(* CODESYS project Elevator_student_1.project

Project tree, tasks and I/O mapping:
  Device : CODESYS Control Win V3, 3S - Smart Software Solutions GmbH, version 3.5.17.10
    application Application
      libraries: Standard, * (System); VisuDialogs, * (System); Util, * (System)
      task MainTask (cyclic, interval t#10ms, priority 1) calls Model, PLC_PRG
      program Model [ST]
      visualisation Visualization
      global variables GVL
      program PLC_PRG [ST]
      function block StartMotor [ST]
      function block DoorOpenClose [FBD]
  text list GlobalTextList
*)

// Device/Application/GVL
VAR_GLOBAL
	// Sensors:
	onfloor0:BOOL;		// Elevator at floor 0
	onfloor1:BOOL;		// Elevator at floor 1
	onfloor2:BOOL;		// Elevator at floor 2
	doorclosed0:BOOL;	// Doors at floor 0 are closed
	doorclosed1:BOOL;	// Doors at floor 1 are closed
	doorclosed2:BOOL;	// Doors at floor 2 are closed *)
	button0:BOOL;		// Call button at floor 0
	button1:BOOL;		// Call button at floor 1
	button2:BOOL;		// Call button at floor 2
	call0:BOOL;			// Request floor 0 from inside the cabin 
	call1:BOOL;			// Request floor 1 from inside the cabin
	call2:BOOL;			// Request floor 2 from inside the cabin
	
	// Actuators:
	up:BOOL;			// Control the elevator to go up
	down:BOOL;			// Control the elevator to go down
	open0:BOOL;			// Open the doors at floor 0
	open1:BOOL;			// Open the doors at floor 1
	open2:BOOL;			// Open the doors at floor 2
	
	// Other variables:
	go:BOOL;
	x:INT;				// Next destination floor number
END_VAR

// Device/Application/Model
PROGRAM Model

VAR CONSTANT
	// Define following variables as required
	maxSpeedLift :REAL := 0.5;
	accLift :REAL := 0.25;
	speedDoor :REAL := 0.5;
	cycleTime :DWORD := 10;
END_VAR

VAR
	// Following variables are inputs to the model
	motorUp :BOOL;
	motorDown :BOOL;
	door0 :BOOL;
	door1 :BOOL;
	door2 :BOOL;
	///////////////////////////////////////////////
	// Following variables are outpus from the model
	buttonFloor0: BOOL;
	buttonFloor1: BOOL;
	buttonFloor2: BOOL;
	requestFloor0 :BOOL;
	requestFloor1 :BOOL;
	requestFloor2 :BOOL;
	elevatorAtFloor0 :BOOL;
	elevatorAtFloor1 :BOOL;
	elevatorAtFloor2 :BOOL;
	door0Closed :BOOL;
	door1Closed :BOOL;
	door2Closed :BOOL;
	////////////////////////////////////////////
	elevatorPos :REAL :=30.0;
	speedLift :REAL := 0.0;
	doIntegral :INTEGRAL;
	door0LeftPos :REAL :=0.0;
	door0RightPos :REAL :=0.0;
	door1LeftPos :REAL :=0.0;
	door1RightPos :REAL :=0.0;
	door2LeftPos :REAL :=0.0;
	door2RightPos :REAL :=0.0;
	elevatorAtFloor :INT :=2;
	floor0 :BOOL;
	floor1 :BOOL;
	floor2 :BOOL;
	heightSensor :REAL := 0.0; // Output the height of the cabin.
END_VAR

// Definition of the inputs to the model, which correspond to the outputs from the controller.
motorUp := GVL.up;
motorDown := GVL.down;
door0 := GVL.open0;
door1 := GVL.open1;
door2 := GVL.open2;

// Control of the elevator
// First calculate its speed
IF motorUp OR motorDown THEN
	doIntegral(IN:=accLift,TM:=cycleTime,RESET:= NOT(motorUp OR motorDown),OUT=>speedLift);
ELSE
	doIntegral(RESET:=TRUE);
	speedLift := 0.0;
END_IF
// Limit the speed
IF (speedLift > maxSpeedLift) THEN
	speedLift := maxSpeedLift;
END_IF

// Then apply the speed if commanded
IF motorUp AND elevatorPos > 0.0 THEN
	elevatorPos := elevatorPos - speedLift;
END_IF

IF motorDown AND elevatorPos < 440.0 THEN
	elevatorPos := elevatorPos + speedLift;
END_IF

// Control of doors at floor 0. Doors are mirrored
IF door0 AND door0LeftPos > -50.0 THEN
	door0LeftPos := door0LeftPos - speedDoor;
	door0RightPos := - door0LeftPos;
END_IF
IF NOT(door0) AND door0LeftPos < 0.0 THEN
	door0LeftPos := door0LeftPos + speedDoor;
	door0RightPos := - door0LeftPos;
END_IF

// Control of doors at floor 1
IF door1 AND door1LeftPos > -50.0 THEN
	door1LeftPos := door1LeftPos - speedDoor;
	door1RightPos := - door1LeftPos;
END_IF
IF NOT(door1) AND door1LeftPos < 0.0 THEN
	door1LeftPos := door1LeftPos + speedDoor;
	door1RightPos := - door1LeftPos;
END_IF

// Control of doors at floor 2
IF door2 AND door2LeftPos > -50.0 THEN
	door2LeftPos := door2LeftPos - speedDoor;
	door2RightPos := - door2LeftPos;
END_IF
IF NOT(door2) AND door2LeftPos < 0.0 THEN
	door2LeftPos := door2LeftPos + speedDoor;
	door2RightPos := - door2LeftPos;
END_IF

// Status sensors whether the doors are closed or not
IF door0LeftPos < 0.0 THEN
	door0Closed := FALSE;
ELSE
	door0Closed := TRUE;
END_IF
IF door1LeftPos < 0.0 THEN
	door1Closed := FALSE;
ELSE
	door1Closed := TRUE;
END_IF
IF door2LeftPos < 0.0 THEN
	door2Closed := FALSE;
ELSE
	door2Closed := TRUE;
END_IF

// Determine floor number of elevator
IF elevatorPos < 30.5 THEN
	elevatorAtFloor := 2;
	elevatorAtFloor2 := TRUE;
	elevatorAtFloor0 := FALSE;
	elevatorAtFloor1 := FALSE;
ELSIF (elevatorPos  > 224.5) AND (elevatorPos < 225.5) THEN
	elevatorAtFloor := 1;
	elevatorAtFloor1 := TRUE;
	elevatorAtFloor0 := FALSE;
	elevatorAtFloor2 := FALSE;
ELSIF elevatorPos > 418.5 THEN
	elevatorAtFloor := 0;
	elevatorAtFloor0 := TRUE;
	elevatorAtFloor1 := FALSE;
	elevatorAtFloor2 := FALSE;
ELSE
	elevatorAtFloor2 := FALSE;
	elevatorAtFloor0 := FALSE;
	elevatorAtFloor1 := FALSE;	
END_IF

// Used to mantain the buttons state (visuzalization is a tap, hence a flip/flop is
// implemented here in order to mantain the status of the button and the "light".
IF floor0 THEN
	buttonFloor0 := TRUE;
END_IF
IF floor1 THEN
	buttonFloor1 := TRUE;
END_IF
IF floor2 THEN
	buttonFloor2 := TRUE;
END_IF

// Reset function for the request button. If the cabin is at the same floor and doors are opened,
// reset request of the floor
IF (requestFloor0 OR buttonFloor0) AND elevatorAtFloor0 AND (door0LeftPos < -49.5) THEN
	requestFloor0 := FALSE;
	buttonFloor0 := FALSE;
END_IF
IF (requestFloor1 OR buttonFloor1) AND elevatorAtFloor1 AND (door1LeftPos < -49.5) THEN
	requestFloor1 := FALSE;
	buttonFloor1 := FALSE;
END_IF
IF (requestFloor2 OR buttonFloor2) AND elevatorAtFloor2 AND (door2LeftPos < -49.5) THEN
	requestFloor2 := FALSE;
	buttonFloor2 := FALSE;
END_IF

// Extra functionality: the following code provides the reading of an analog sensor measuring the 
// height position of the elevator. It ouputs a value between 0..2 in normal conditions (i.e. the
// elevator does not go below o or over 2). If the elevator is driven below ground level, a minus
// sign number will be output. In case the elevator is driven over the second floor, a number
// higher than 2.0 will be output.
heightSensor := (419.0 - elevatorPos) / 389.0 * 2;

// Lastly, update outputs from the model, which correspond to the inputs of the controller.
GVL.button0 := buttonFloor0;
GVL.button1 := buttonFloor1;
GVL.button2 := buttonFloor2;
GVL.call0 := requestFloor0;
GVL.call1 := requestFloor1;
GVL.call2 := requestFloor2;
GVL.onfloor0 := elevatorAtFloor0;
GVL.onfloor1 := elevatorAtFloor1;
GVL.onfloor2 := elevatorAtFloor2;
GVL.doorclosed0 := door0Closed;
GVL.doorclosed1 := door1Closed;
GVL.doorclosed2 := door2Closed;

END_PROGRAM

// Device/Application/PLC_PRG
PROGRAM PLC_PRG
VAR
	startMoving:StartMotor;
	openClose:DoorOpenClose;
END_VAR

// Järjestelmätoiminto 1
gvl.go := TRUE;	// Yksikkötestausta varten
x := 0;			// Yksikkötestausta varten

WHILE gvl.go DO
	IF (gvl.onfloor0 AND x = 0) OR (gvl.onfloor1 AND x = 1) OR (gvl.onfloor2 AND x = 2) THEN;
		CASE gvl.x OF
		0:	gvl.open0 := TRUE;
			openClose();
			openClose.trigger := TRUE;
			gvl.open0 := openClose.output;
			
		1:	gvl.open1 := TRUE;
			openClose();
			openClose.trigger := TRUE;
			gvl.open1 := openClose.output;
			
		2:	gvl.open2 := TRUE;
			openClose();
			openClose.trigger := TRUE;
			gvl.open2 := openClose.output;
		END_CASE
		gvl.go := FALSE;
		RETURN;
	END_IF
	
	startMoving();
	Model();

	IF (NOT x = 1) AND gvl.onfloor1 AND (gvl.button1 OR gvl.call1) THEN
		gvl.up := FALSE;
		gvl.down := FALSE;
		gvl.open1 := TRUE;
		openClose();
		openClose.trigger := TRUE;
		gvl.open1 := openClose.output;
		gvl.call1 := FALSE;
		gvl.button1 := FALSE;
		startMoving();
		Model();
		openClose.trigger := FALSE;
	END_IF
		
	IF (x = 0 AND gvl.onfloor0) OR (x = 1 AND gvl.onfloor1) OR (x = 2 AND gvl.onfloor2) THEN
		gvl.up := FALSE;
		gvl.down := FALSE;
		CASE gvl.x OF
		0:	gvl.open0 := TRUE;
			openClose();
			openClose.trigger := TRUE;
			gvl.open0 := openClose.output;
			
		1:	gvl.open1 := TRUE;
			openClose();
			openClose.trigger := TRUE;
			gvl.open1 := openClose.output;
			
		2:	gvl.open2 := TRUE;  
			openClose();
			openClose.trigger := TRUE;
			gvl.open2 := openClose.output;	
		END_CASE
		gvl.go := FALSE;
	END_IF
	
	openClose.trigger := FALSE;
END_WHILE

END_PROGRAM

// Device/Application/StartMotor
FUNCTION_BLOCK StartMotor

IF gvl.onfloor0 AND (x = 1 OR x = 2) THEN;
	gvl.up := TRUE;
ELSIF gvl.onfloor2 AND (x = 0 OR x = 1) THEN;
	gvl.down := TRUE;
ELSIF gvl.onfloor1 AND x = 0 THEN;
	gvl.down := TRUE;
ELSIF gvl.onfloor1 AND x = 2 THEN;
	gvl.up := TRUE;
END_IF

END_FUNCTION_BLOCK

// Device/Application/DoorOpenClose
FUNCTION_BLOCK DoorOpenClose
VAR_INPUT
	trigger: BOOL;
	delay: TIME := T#1.5S;
END_VAR
VAR_OUTPUT
	elapsed: TIME;
	output: BOOL;
END_VAR
VAR
	OpenClose: TOF;
END_VAR
VAR // added by the converter: edge detectors and wires of the graphical bodies
    _rt1 : R_TRIG;
END_VAR

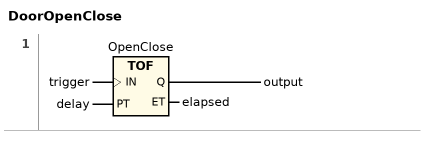
// NETWORK 1
_rt1(CLK := trigger);
OpenClose(IN := _rt1.Q, PT := delay, ET => elapsed); // TOF
output := OpenClose.Q;

END_FUNCTION_BLOCK

// Device/Application/Visualization
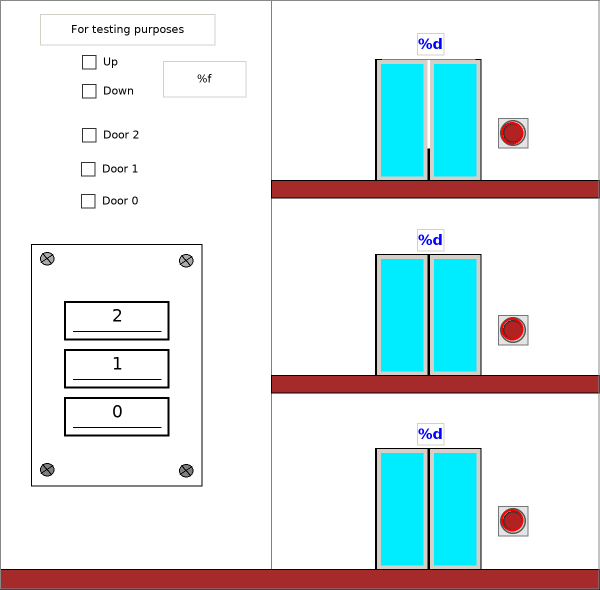
VISUALIZATION Visualization  // 600x590
    Rectangle (347,2 171x585)
    RoundedRectangle (31,244 171x242)
    Rectangle (380,30 97x120)
        p2738717112: Model.elevatorPos
    Rectangle (430,60 50x120)
        p3560616238: Model.door2RightPos
    Rectangle (377,60 50x120)
        p3560616238: Model.door2LeftPos
    Rectangle (377,255 50x120)
        p3560616238: Model.door1LeftPos
    Rectangle (430,255 50x120)
        p3560616238: Model.door1RightPos
    Rectangle (377,449 50x120)
        p3560616238: Model.door0LeftPos
    Rectangle (430,449 50x120)
        p3560616238: Model.door0RightPos
    RoundedRectangle (64,397 105x39)
        OnMouseDown: execute { Model.requestFloor0 := TRUE; }
    Label (87,400 61x23), "0"
    Line (73,427) (161,427)
    RoundedRectangle (64,349 105x39)
        OnMouseDown: execute { Model.requestFloor1 := TRUE; }
    Label (87,352 61x23), "1"
    Line (73,379) (161,379)
    RoundedRectangle (64,301 105x39)
        OnMouseDown: execute { Model.requestFloor2 := TRUE; }
    Label (87,304 61x23), "2"
    Line (73,331) (161,331)
    Line (73,427) (161,427), invisible if: NOT(Model.requestFloor0)
    Line (73,379) (161,379), invisible if: NOT(Model.requestFloor1)
    Line (73,331) (161,331), invisible if: NOT(Model.requestFloor2)
    Ellipse (40,463 14x13)
    Line (42,464) (51,474)
    Line (41,473) (53,465)
    Ellipse (179,254 14x13)
    Line (181,255) (190,265)
    Line (180,264) (192,256)
    Ellipse (40,252 14x13)
    Line (42,253) (51,263)
    Line (41,262) (53,254)
    Ellipse (179,464 14x13)
    Line (181,465) (190,475)
    Line (180,474) (192,466)
    Rectangle (271,180 329x18)
    Rectangle (271,375 329x18)
    Polygon (271,180) (375,180) (375,59) (481,59) (481,180) (600,180) (600,0) (271,0)
    Polygon (271,569) (375,569) (375,448) (481,448) (481,569) (600,569) (600,393) (271,393)
    Polygon (271,375) (375,375) (375,254) (481,254) (481,375) (600,375) (600,198) (271,198)
    PushSwitch (498,118 30x30), variable: Model.floor2, behaviour: TAP, style: Switch-PushSwitch-Red
    Textfield (417,423 27x22), "%d", text variable: Model.elevatorAtFloor
    Textfield (417,229 27x22), "%d", text variable: Model.elevatorAtFloor
    PushSwitch (498,506 30x30), variable: Model.floor0, behaviour: TAP, style: Switch-PushSwitch-Red
    PushSwitch (498,315 30x30), variable: Model.floor1, behaviour: TAP, style: Switch-PushSwitch-Red
    Ellipse (501,509 22x22), invisible if: NOT(Model.buttonFloor0)
    Ellipse (501,318 22x22), invisible if: NOT(Model.buttonFloor1)
    Ellipse (501,122 22x22), invisible if: NOT(Model.buttonFloor2)
    Textfield (417,33 27x22), "%d", text variable: Model.elevatorAtFloor
    Rectangle (0,569 600x21)
    Checkbox (80,47 57x30), "Up", variable: GVL.up
    Checkbox (80,76 78x30), "Down", variable: GVL.down
    Checkbox (79,186 79x30), "Door 0", variable: GVL.open0
    Checkbox (79,154 79x30), "Door 1", variable: GVL.open1
    Checkbox (80,120 80x30), "Door 2", variable: GVL.open2
    Textfield (40,14 175x31), "For testing purposes"
    Textfield (163,61 83x36), "%f", text variable: Model.heightSensor
END_VISUALIZATION
